FUNCTION_BLOCK FB_Base

F_IsSystemValid();

END_FUNCTION_BLOCK

(* stored: Version 1.1.0.1, ProductVersion 3.1.4024.12
   POU FB_Base: Id {00104c86-c6f6-0cc6-3725-ac227baa1029}, SpecialFunc None *)
